{attribute addProperty BoxType "KL8524"}
{attribute addProperty Id "Channel_1Channel_98BE1B6E00"}
{attribute addProperty CRC "3861074838"}
{attribute addProperty SizeInBites "0"}
{attribute addProperty SizeInBytes "0"}
TYPE KL8524_E6235396 :
STRUCT
	{attribute addProperty Name "Channel_1"}
	Channel_1 : Channel_98BE1B6E;
END_STRUCT
END_TYPE

(* stored: Version 1.2.0.0, ProductVersion 3.1.4024.9
   DUT KL8524_E6235396: Id {b833b96a-dc0b-4b6c-97ab-7c175ed78a01} *)
